FUNCTION_BLOCK FB_NetContactor_IO
VAR
	b_Write					AT %Q* : ARRAY[1..2] OF BOOL;	
	b_Read					AT %I* : ARRAY[1..3] OF BOOL;
END_VAR

VAR_INPUT
	b_RotationSelect					: BOOL := 0; //0: Clockwise, 1: Anti-Clockwise
	b_ForceCloseCommand					: BOOL := 0; //O; Open, 1:close
END_VAR

VAR_IN_OUT
	get								: ST_Netcontactor_get;
	b_NetcontEDM					: BOOL;
END_VAR
VAR
END_VAR

read();
Write();

METHOD PRIVATE Read
get.b_NetcontRightFb 	:= b_read[1];
get.b_NetcontLeftFb		:= b_read[2];
b_NetcontEDM			:= b_read[3];
END_METHOD

METHOD PRIVATE Write

VAR_INST
	
END_VAR
b_Write[1] := b_RotationSelect;
b_Write[2] := b_ForceCloseCommand;
END_METHOD

END_FUNCTION_BLOCK

(* stored: Version 1.1.0.1, ProductVersion 3.1.4026.18
   POU FB_NetContactor_IO: Id {4356f18b-f1a8-4cd8-ab67-3b8eff04dfda}, SpecialFunc None
   Method Read: Id {b07212c0-ccce-4d23-9a4c-59e59afc1434}
   Method Write: Id {edf143f9-d2e8-4f29-97a7-35116a7d9899} *)
